// TwinCAT 3 PLC project PLC
// ProgramVersion: 3.1.4026.20
// libraries:
//   Tc2_Standard, * (Beckhoff Automation GmbH)
//   Tc2_System, * (Beckhoff Automation GmbH)
//   Tc2_Utilities, * (Beckhoff Automation GmbH)
// project tree:
//   DUTs/ ST_LrealDataPoint.TcDUT
//   / PlcTask.TcTTO
//   POUs/ FB_FifoIndexer.TcPOU, FB_LowPassFilter.TcPOU, FB_Scheduler.TcPOU, MAIN.TcPOU
// real-time tasks:
//   TASK PlcTask: cycle T#10ms, priority 20, ADS port 350

CONFIGURATION PLC
    RESOURCE PLC ON TwinCAT3
        TASK PlcTask(INTERVAL := T#10ms, PRIORITY := 20);
        PROGRAM MAIN WITH PlcTask : MAIN;
    END_RESOURCE
END_CONFIGURATION

// ---- DUTs/ST_LrealDataPoint.TcDUT
TYPE ST_LrealDataPoint :
STRUCT
	Timestamp	: ULINT;
	Value		: LREAL;
END_STRUCT
END_TYPE

// ---- POUs/MAIN.TcPOU
PROGRAM MAIN
VAR_INPUT
{attribute 'HMEye':='200'}
	StartCommand	: BOOL;
	
{attribute 'HMEye':='200'}
	StopCommand		: BOOL;
END_VAR

VAR_OUTPUT
{attribute 'HMEye':='1000'}
{attribute 'IsReadOnly':='true'}
	CurrentDT		: DT;
	
{attribute 'HMEye':='1000'}
	Activity		: BOOL;
	
{attribute 'HMEye':='200'}
	Percent			: LREAL;
	
{attribute 'HMEye':='5000'} 
	PercentHistory	: ARRAY[0..9] OF ST_LrealDataPoint;
END_VAR
VAR
	_raw		: LREAL;
	_scaled		: LREAL;
	_enable		: BOOL;
	_dequeue	: BOOL;
	_reset		: BOOL;
	
	fbLowPass	: FB_LowPassFilter;
	fbScheduler	: FB_Scheduler;
	fbRand		: DRAND;
	fbFifo		: FB_FifoIndexer := (MaxSize := 10, EnableWrapAround := TRUE);
	
END_VAR
VAR CONSTANT
	EPOCH_DT	: DT := DT#1970-01-01-00:00:00;
END_VAR

fbScheduler();
fbLowPass(Enable := _enable, Raw := _scaled, TimeConstant := 5, CycleTime := 0.01, Filtered => Percent);
CurrentDT := fbScheduler.CurrentDT;

_enable S= StartCommand;
_enable R= StopCommand;
StartCommand := StopCommand := FALSE;

IF fbScheduler.Every1Second THEN
	Activity := NOT Activity;
END_IF

IF fbScheduler.Every5Seconds THEN
	IF _enable THEN
		PercentHistory[fbFifo.WriteIndex].Timestamp := DT_TO_FILETIME64(fbScheduler.CurrentDT);
		PercentHistory[fbFifo.WriteIndex].Value := Percent;
		fbFifo.Enqueue();
    END_IF
END_IF

IF fbScheduler.Every10Seconds THEN
	fbRand(Seed := 0, Num => _raw);
	_scaled := _raw * 100;
END_IF

IF _dequeue AND NOT fbFifo.IsEmpty THEN
	PercentHistory[fbFifo.ReadIndex].Timestamp := DT_TO_FILETIME64(EPOCH_DT);
	PercentHistory[fbFifo.ReadIndex].Value := 0;
	fbFifo.Dequeue();
	_dequeue := FALSE;
END_IF

END_PROGRAM

// ---- POUs/FB_LowPassFilter.TcPOU
FUNCTION_BLOCK FB_LowPassFilter
VAR_INPUT
	Enable			: BOOL;
    Raw				: LREAL; // Raw input signal
    TimeConstant	: LREAL; // Smoothing time constant (seconds)
    CycleTime		: LREAL; // PLC cycle time (seconds)
END_VAR
VAR_OUTPUT
    Filtered		: LREAL; // Current filtered value
END_VAR
VAR
    _lastFiltered	: LREAL; // Previous filtered value
    _alpha			: LREAL; // Smoothing factor
    _initialized	: BOOL;
END_VAR

IF Enable THEN
	IF NOT _initialized THEN
		_lastFiltered := Raw; // Initialize to raw value
		Filtered := Raw;
		_initialized := TRUE;
	END_IF;
	
	IF TimeConstant <= 0.0 OR CycleTime <= 0.0 THEN
		Filtered := _lastFiltered; // No update if invalid inputs
	ELSE
		_alpha := CycleTime / TimeConstant;
		Filtered := _lastFiltered + _alpha * (Raw - _lastFiltered);
		_lastFiltered := Filtered; // Update for next cycle
	END_IF;
END_IF

END_FUNCTION_BLOCK

// ---- POUs/FB_Scheduler.TcPOU
FUNCTION_BLOCK FB_Scheduler
VAR_INPUT
END_VAR
VAR_OUTPUT
	Every1Second	: BOOL; // TRUE for one cycle every 1 seconds
    Every5Seconds	: BOOL; // TRUE for one cycle every 5 seconds
    Every10Seconds	: BOOL; // TRUE for one cycle every 10 seconds
    Every20Seconds	: BOOL; // TRUE for one cycle every 30 seconds
    Every30Seconds	: BOOL; // TRUE for one cycle every 30 seconds
    Every1Minutes	: BOOL; // TRUE for one cycle every 1 minutes
    Every2Minutes	: BOOL; // TRUE for one cycle every 2 minutes
    Every5Minutes	: BOOL; // TRUE for one cycle every 5 minutes
	CurrentDT		: DT;
	CurrentUTC		: DT;
END_VAR
VAR
    _lastTrigger1	: DT;
    _lastTrigger5	: DT;
    _lastTrigger10	: DT;
	_lastTrigger20	: DT;
	_lastTrigger30	: DT;
	_lastTrigger60	: DT;
	_lastTrigger120	: DT;
	_lastTrigger300	: DT;
    _elapsed		: LREAL; // Elapsed time since last trigger (seconds)
    _initialized	: BOOL;
	fbSysTime		: FB_LocalSystemTime := (bEnable := TRUE, dwCycle := 1);
    fbTzInfo        : FB_GetTimeZoneInformation := (bExecute := TRUE);
    fbTzToUtc       : FB_TzSpecificLocalTimeToSystemTime;
END_VAR

fbSysTime();
fbTzInfo();
fbTzToUtc(in := fbSysTime.systemTime, tzInfo := fbTzInfo.tzInfo);
CurrentDT := SYSTEMTIME_TO_DT(fbSysTime.systemTime);
CurrentUTC := SYSTEMTIME_TO_DT(fbTzToUtc.out);

IF NOT _initialized THEN
    _lastTrigger1	:= CurrentDT;
    _lastTrigger5	:= CurrentDT;
    _lastTrigger10	:= CurrentDT;
    _lastTrigger20	:= CurrentDT;
    _lastTrigger30	:= CurrentDT;
    _lastTrigger60	:= CurrentDT;
    _lastTrigger120	:= CurrentDT;
    _lastTrigger300	:= CurrentDT;
    _initialized := TRUE;
END_IF;

_elapsed := TO_LREAL(CurrentDT - _lastTrigger1) / 1000.0;
IF _elapsed >= 1.0 THEN
	Every1Second := TRUE;
	_lastTrigger1 := CurrentDT;
ELSE
	Every1Second := FALSE;
END_IF;

_elapsed := TO_LREAL(CurrentDT - _lastTrigger5) / 1000.0;
IF _elapsed >= 5.0 THEN
	Every5Seconds := TRUE;
	_lastTrigger5 := CurrentDT;
ELSE
    Every5Seconds := FALSE;
END_IF;

_elapsed := TO_LREAL(CurrentDT - _lastTrigger10) / 1000.0;
IF _elapsed >= 10.0 THEN
    Every10Seconds := TRUE;
    _lastTrigger10 := CurrentDT;
ELSE
    Every10Seconds := FALSE;
END_IF;

_elapsed := TO_LREAL(CurrentDT - _lastTrigger20) / 1000.0;
IF _elapsed >= 20.0 THEN
    Every20Seconds := TRUE;
    _lastTrigger20 := CurrentDT;
ELSE
    Every20Seconds := FALSE;
END_IF;

_elapsed := TO_LREAL(CurrentDT - _lastTrigger30) / 1000.0;
IF _elapsed >= 30.0 THEN
    Every30Seconds := TRUE;
    _lastTrigger30 := CurrentDT;
ELSE
    Every30Seconds := FALSE;
END_IF;

_elapsed := TO_LREAL(CurrentDT - _lastTrigger60) / 1000.0;
IF _elapsed >= 60.0 THEN
    Every1Minutes := TRUE;
    _lastTrigger60 := CurrentDT;
ELSE
    Every1Minutes := FALSE;
END_IF;

_elapsed := TO_LREAL(CurrentDT - _lastTrigger120) / 1000.0;
IF _elapsed >= 120.0 THEN
    Every2Minutes := TRUE;
    _lastTrigger120 := CurrentDT;
ELSE
    Every2Minutes := FALSE;
END_IF;

_elapsed := TO_LREAL(CurrentDT - _lastTrigger300) / 1000.0;
IF _elapsed >= 300.0 THEN
    Every5Minutes := TRUE;
    _lastTrigger300 := CurrentDT;
ELSE
    Every5Minutes := FALSE;
END_IF;

END_FUNCTION_BLOCK

// ---- POUs/FB_FifoIndexer.TcPOU
FUNCTION_BLOCK FB_FifoIndexer
VAR_INPUT
    MaxSize : UDINT;  // Set once, e.g., in init
	EnableWrapAround : BOOL := FALSE;	// Enable wrap-around when buffer is full
END_VAR
VAR_OUTPUT
END_VAR
VAR
    _readIndex : UDINT := 0;
    _writeIndex : UDINT := 0;
    _count : UDINT := 0;
END_VAR

PROPERTY Count : UDINT
GET
Count := _count;
END_GET
END_PROPERTY

METHOD Dequeue : BOOL;
VAR_INPUT
END_VAR
IF IsEmpty THEN 
	Dequeue := FALSE; // Empty
	RETURN;
END_IF

Dequeue := TRUE;
_readIndex := (_readIndex + 1) MOD MaxSize;
_count := _count - 1;
END_METHOD

METHOD Enqueue : BOOL;
VAR_INPUT
END_VAR
IF IsFull AND NOT EnableWrapAround THEN
	Enqueue := FALSE; // Full
	RETURN;
END_IF

Enqueue := TRUE;
_writeIndex := (_writeIndex + 1) MOD MaxSize;
_count := _count + 1;
END_METHOD

PROPERTY IsEmpty : BOOL
GET
IsEmpty := (_readIndex = _writeIndex) AND (_count = 0);
END_GET
END_PROPERTY

PROPERTY IsFull : BOOL
GET
IsFull := _writeIndex = _readIndex AND _count = MaxSize;
END_GET
END_PROPERTY

PROPERTY ReadIndex : UDINT
GET
ReadIndex := _readIndex;
END_GET
END_PROPERTY

PROPERTY WriteIndex : UDINT
GET
WriteIndex := _writeIndex;
END_GET
END_PROPERTY

END_FUNCTION_BLOCK
